// Mitsubishi GX Works2 project: EX04   PLC: Q03UD

PROGRAM Lane1
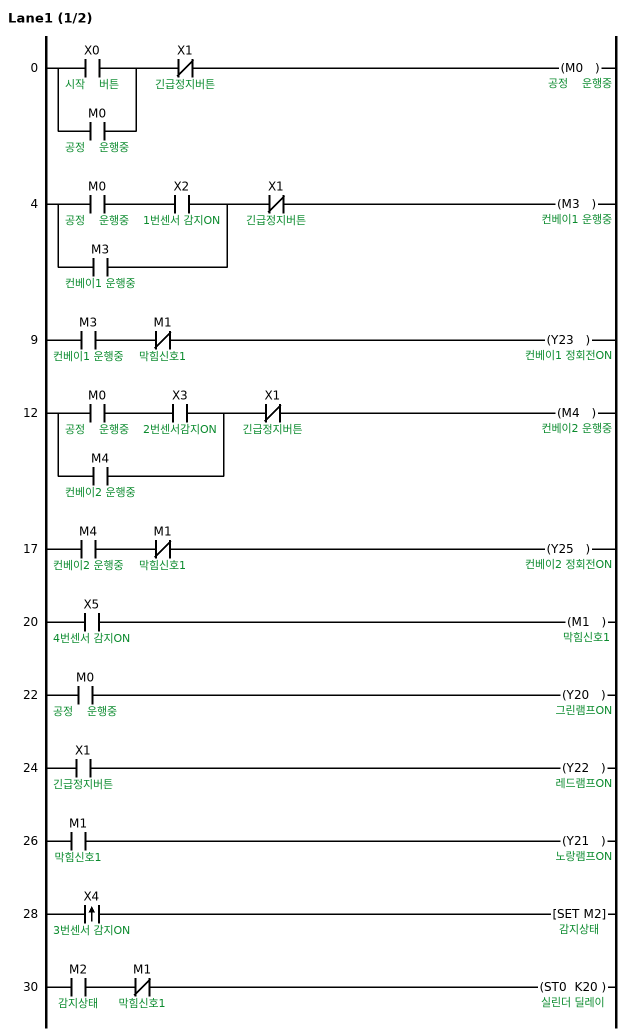
0     LD      X0  ; 시작    버튼
      OR      M0  ; 공정    운행중
      ANI     X1  ; 긴급정지버튼
      OUT     M0  ; 공정    운행중
4     LD      M0  ; 공정    운행중
      AND     X2  ; 1번센서 감지ON
      OR      M3  ; 컨베이1 운행중
      ANI     X1  ; 긴급정지버튼
      OUT     M3  ; 컨베이1 운행중
9     LD      M3  ; 컨베이1 운행중
      ANI     M1  ; 막힘신호1
      OUT     Y23  ; 컨베이1 정회전ON
12    LD      M0  ; 공정    운행중
      AND     X3  ; 2번센서감지ON
      OR      M4  ; 컨베이2 운행중
      ANI     X1  ; 긴급정지버튼
      OUT     M4  ; 컨베이2 운행중
17    LD      M4  ; 컨베이2 운행중
      ANI     M1  ; 막힘신호1
      OUT     Y25  ; 컨베이2 정회전ON
20    LD      X5  ; 4번센서 감지ON
      OUT     M1  ; 막힘신호1
22    LD      M0  ; 공정    운행중
      OUT     Y20  ; 그린램프ON
24    LD      X1  ; 긴급정지버튼
      OUT     Y22  ; 레드램프ON
26    LD      M1  ; 막힘신호1
      OUT     Y21  ; 노랑램프ON
28    LDP     X4  ; 3번센서 감지ON
      SET     M2  ; 감지상태
30    LD      M2  ; 감지상태
      ANI     M1  ; 막힘신호1
      OUT     ST0 K20  ; 실린더 딜레이
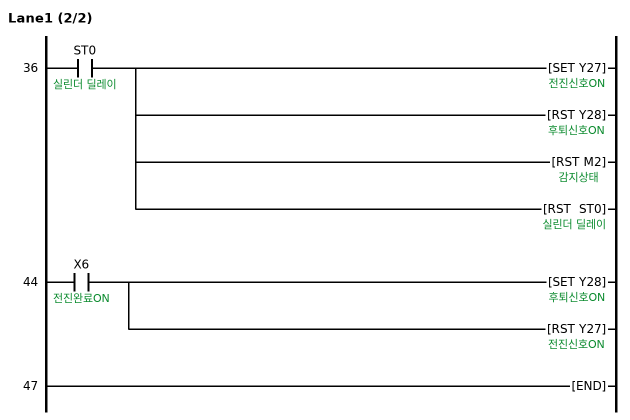
36    LD      ST0  ; 실린더 딜레이
      SET     Y27  ; 전진신호ON
      RST     Y28  ; 후퇴신호ON
      RST     M2  ; 감지상태
      RST     ST0  ; 실린더 딜레이
44    LD      X6  ; 전진완료ON
      SET     Y28  ; 후퇴신호ON
      RST     Y27  ; 전진신호ON
47    END
END_PROGRAM

PROGRAM Lane2
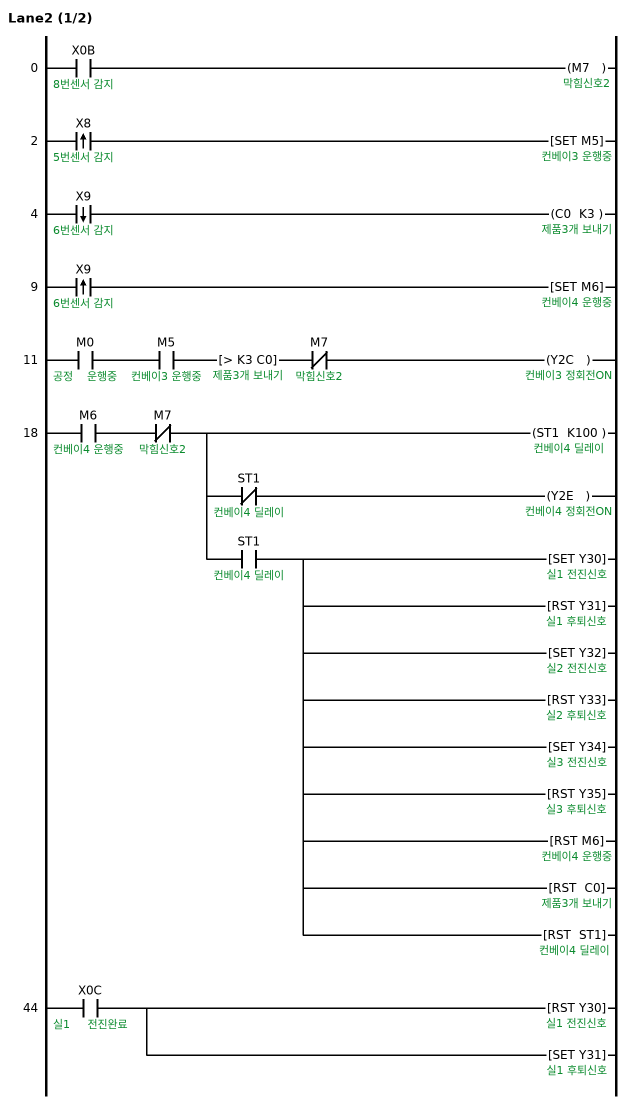
0     LD      X0B  ; 8번센서 감지
      OUT     M7  ; 막힘신호2
2     LDP     X8  ; 5번센서 감지
      SET     M5  ; 컨베이3 운행중
4     LDF     X9  ; 6번센서 감지
      OUT     C0 K3  ; 제품3개 보내기
9     LDP     X9  ; 6번센서 감지
      SET     M6  ; 컨베이4 운행중
11    LD      M0  ; 공정    운행중
      AND     M5  ; 컨베이3 운행중
      AND>    K3 C0  ; 제품3개 보내기
      ANI     M7  ; 막힘신호2
      OUT     Y2C  ; 컨베이3 정회전ON
18    LD      M6  ; 컨베이4 운행중
      ANI     M7  ; 막힘신호2
      OUT     ST1 K100  ; 컨베이4 딜레이
      MPS
      ANI     ST1  ; 컨베이4 딜레이
      OUT     Y2E  ; 컨베이4 정회전ON
      MPP
      AND     ST1  ; 컨베이4 딜레이
      SET     Y30  ; 실1 전진신호
      RST     Y31  ; 실1 후퇴신호
      SET     Y32  ; 실2 전진신호
      RST     Y33  ; 실2 후퇴신호
      SET     Y34  ; 실3 전진신호
      RST     Y35  ; 실3 후퇴신호
      RST     M6  ; 컨베이4 운행중
      RST     C0  ; 제품3개 보내기
      RST     ST1  ; 컨베이4 딜레이
44    LD      X0C  ; 실1     전진완료
      RST     Y30  ; 실1 전진신호
      SET     Y31  ; 실1 후퇴신호
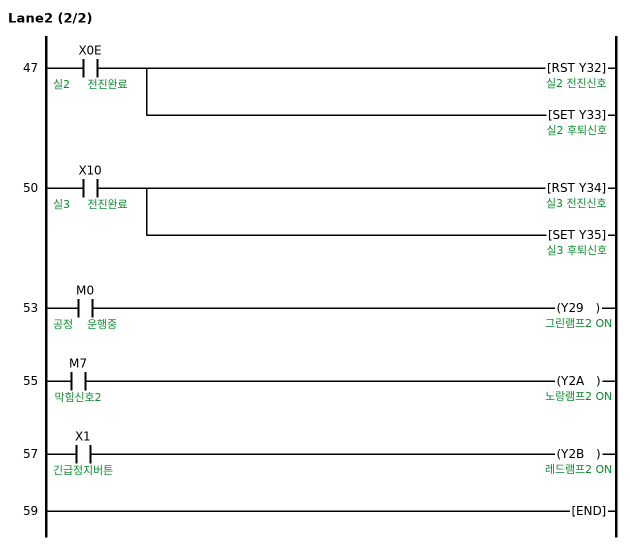
47    LD      X0E  ; 실2     전진완료
      RST     Y32  ; 실2 전진신호
      SET     Y33  ; 실2 후퇴신호
50    LD      X10  ; 실3     전진완료
      RST     Y34  ; 실3 전진신호
      SET     Y35  ; 실3 후퇴신호
53    LD      M0  ; 공정    운행중
      OUT     Y29  ; 그린램프2 ON
55    LD      M7  ; 막힘신호2
      OUT     Y2A  ; 노랑램프2 ON
57    LD      X1  ; 긴급정지버튼
      OUT     Y2B  ; 레드램프2 ON
59    END
END_PROGRAM

// device comments not shown above
X7  ; 전진완료신호
X0D  ; 실1     후퇴완료
X0F  ; 실2     후퇴완료
X11  ; 실3     후퇴완료
Y10  ; 그린램프ON
Y11  ; 노랑램프ON
Y12  ; 레드램프ON
Y13  ; 컨베이1 정회전ON
Y15  ; 컨베이2 정회전ON
Y17  ; 전진신호ON
Y18  ; 후퇴신호ON
Y1C  ; 컨베이3 정회전ON
Y2D  ; 컨베이4 정회전ON
T0  ; 실린더 딜레이
T1  ; 컨베이4 딜레이
